FUNCTION MUL3 : REAL
VAR_INPUT
	in1 : REAL;
	in2 : REAL;
	in3 : REAL;
END_VAR
VAR
END_VAR

MUL3 := in1 * in2 * in3;

END_FUNCTION

(* stored: Version 1.1.0.1, ProductVersion 3.1.4024.3
   POU MUL3: Id {e727b9e5-a07b-4ef4-961f-064e412bd7bd}, SpecialFunc None *)
